Fanuc KAREL source: kf00100.KL

PROGRAM KF00100
%STACKSIZE=65535
%PRIORITY=65535
%NOLOCKGROUP
%ENVIRONMENT REGOPE
VAR
I : INTEGER
J : INTEGER
X : REAL
Y : REAL
B : BOOLEAN
C : BOOLEAN
TXT : STRING[80]
TXT2 : STRING[80]
AI : ARRAY[4] OF INTEGER
BI : ARRAY[4] OF INTEGER
P : XYZWPR
JP : JOINTPOS9
PF : POSITION
STATUS : INTEGER
-- UNRESOLVED DECLARATIONS (source type spelling not recovered)
-- V1 : TYPE_0x0013 (type_u16=0x0013)
-- V2 : TYPE_0x0013 (type_u16=0x0013)
BEGIN
I=3
X=2.5
SET_POS_REG(1,P,STATUS,1)
END KF00100
